% RSLogix 500 project Q3.RSS, saved by version 8.30.00.16 %
PROJECT "Q3"    % processor: Bul.1763 MicroLogix 1100 Series B %

PROGRAM FILES
  LAD 2   6 rungs

DATA FILES
  O0 OUTPUT  4 elements
  I1 INPUT  6 elements
  S2 STATUS  66 elements
  B3 BINARY  1 elements
  T4 TIMER  2 elements
  C5 COUNTER  1 elements
  R6 CONTROL  1 elements
  N7 INTEGER  1 elements
  F8 FLOAT  1 elements

LADDER 2
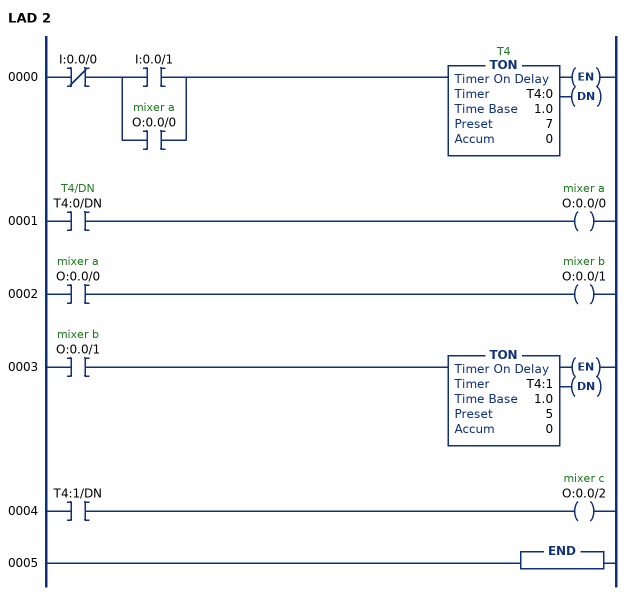
% Rung: 0 %
SOR XIO I:0.0/0 BST XIC I:0.0/1 NXB XIC O:0.0/0 BND TON T4:0 1.0 7 0 EOR
%   O:0.0/0  "mixer a" %
%   T4:0  T4 %
% Rung: 1 %
SOR XIC T4:0/DN OTE O:0.0/0 EOR
%   T4:0  T4 %
%   O:0.0/0  "mixer a" %
% Rung: 2 %
SOR XIC O:0.0/0 OTE O:0.0/1 EOR
%   O:0.0/0  "mixer a" %
%   O:0.0/1  "mixer b" %
% Rung: 3 %
SOR XIC O:0.0/1 TON T4:1 1.0 5 0 EOR
%   O:0.0/1  "mixer b" %
% Rung: 4 %
SOR XIC T4:1/DN OTE O:0.0/2 EOR
%   O:0.0/2  "mixer c" %
% Rung: 5 %
SOR END EOR

DATA TABLE (non-zero values as saved)
DATA T4
% .PRE .ACC %
% T4:0 % 7 0
% T4:1 % 5 0
